(* CODESYS project Intro_to_automation.project

Project tree, tasks and I/O mapping:
  Device : CODESYS Control Win V3 x64, CODESYS, version 3.5.21.30
    application Application
      libraries: Standard, 3.5.18.0 (System)
      task MainTask (cyclic, interval t#20ms, priority 1) calls PLC_PRG
      task VISU_TASK (cyclic, interval 100 ms, priority 31) calls VisuElems.Visu_Prg
      program PLC_PRG [LD]
      visualisation Visualization
  libraries: VisuSymbols, 4.5.0.0 (System)
  visualisation Visualization
  text list GlobalTextList
*)

// Device/Application/PLC_PRG
PROGRAM PLC_PRG
VAR
	Button1: BOOL;
	Bulb1: BOOL;
	Step1: BOOL;
	Step2: BOOL;
	Step3: BOOL;
	Bulb2: BOOL;
	TON_1: TON;
	Time_ET1: TIME;
	TON_2: TON;
	TimeET_2: TIME;
	TimeET_3: TIME;
	TON_3: TON;
	Reset: BOOL;
	EmergencyStop: BOOL;
	Interrupt: BOOL;
END_VAR

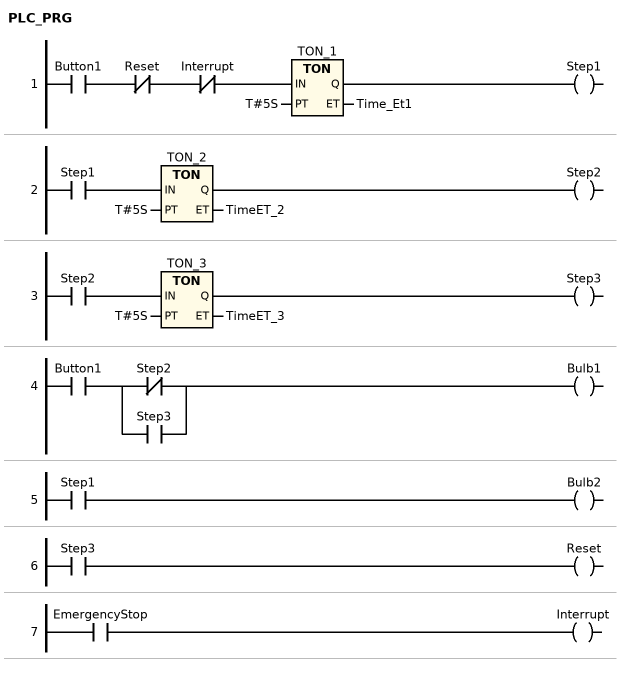
// NETWORK 1
TON_1(IN := Button1 AND NOT Reset AND NOT Interrupt, PT := T#5S, ET => Time_Et1); // TON
Step1 := TON_1.Q;

// NETWORK 2
TON_2(IN := Step1, PT := T#5S, ET => TimeET_2); // TON
Step2 := TON_2.Q;

// NETWORK 3
TON_3(IN := Step2, PT := T#5S, ET => TimeET_3); // TON
Step3 := TON_3.Q;

// NETWORK 4
Bulb1 := Button1 AND (NOT Step2 OR Step3);

// NETWORK 5
Bulb2 := Step1;

// NETWORK 6
Reset := Step3;

// NETWORK 7
Interrupt := EmergencyStop;

END_PROGRAM

// /Visualization
VISUALIZATION Visualization  // 1024x768
END_VISUALIZATION

// Device/Application/Visualization
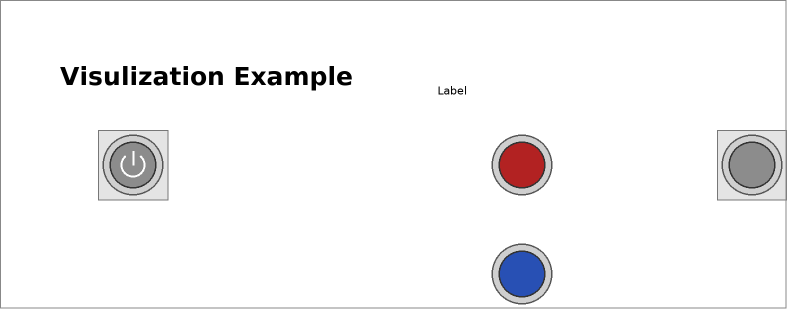
VISUALIZATION Visualization  // 787x309
    Label (160,98 150x30)
    Label (452,91 1x0), "Label"
    Label (67,61 279x30), "Visulization Example"
    PowerSwitch (98,130 70x70), variable: PLC_PRG.Button1, behaviour: TOGGLE, style: Switch-PowerSwitch-Gray
    Lamp1 (487,130 70x70), variable: PLC_PRG.Bulb1, style: Lamp-Lamp1-Red
    Lamp1 (487,239 70x70), variable: PLC_PRG.Bulb2, style: Lamp-Lamp1-Blue
    PushSwitch (717,130 70x70), variable: PLC_PRG.EmergencyStop, behaviour: TOGGLE, style: Switch-PushSwitch-Gray
END_VISUALIZATION
